FUNCTION_BLOCK FB_MonetTelescopeControl IMPLEMENTS I_Telescope
VAR_INPUT
(*
TCS interface section
see https://gitlab.aip.de/bmk10k/telescope_firmware/snippets/5
*)
	bPower				: BOOL;		// true: Power on, false: power off
	bGoHome				: BOOL;		// true: go to home position, unset track/goto if active
	bPark				: BOOL;		// boolean, true: go into park position, ready to stow telescope, unset track/goto
	bTrack				: BOOL;		// boolean, TRUE: MOVE telescope TO last ra/de AND start tracking. Set 'goto' TO FALSE, IF TRUE. FALSE: Stop tracking as soon as possible
	bGoto				: BOOL;		// boolean, TRUE: MOVE telescope TO tau/de AND stop there. Set track TO FALSE, IF TRUE. FALSE: no effect.)	
	bSlew				: BOOL;		// move the telescope to a given az-alt position
	bStop				: BOOL;		// boolean, TRUE: Stop motion OF telescope immediately, set goto AND track TO FALSE. FALSE: Allow motion OF telescope again via track/goto).	
	bReset				: BOOL;		// initiates reset on all axis
	bAutoTrack			: BOOL := TRUE;	// automatic tracking after goto
	fRightAscension		: LREAL := (4.0 + 35.0/60.0 + 54.09/3600.0) *15.0;	// apparent right ascension, degrees, double	
	fDeclination		: LREAL := 16.0 + 30.0/60.0 + 25.4/3600.0;	// apparent declination, degrees, double
	fElevation			: LREAL := 45.0;	// desired elevation of the telescope pointing
	fAzimuth			: LREAL := 320.0;	// desired azimut of the telescope pointing
	fElevationOffset	: LREAL := 0.0;		// absolute offset for elevation
	fAzimuthOffset 		: LREAL := 0.0;		// absolute offset for azimuth
	fTimeOffset			: LREAL := 0.0;		// absolute offset for time
	fDerotatorOffset	: LREAL := 0.0;		// offset for the de-rotator
	
	bEstopTriggered		: BOOL	:= FALSE;	// TODO: CHANGE
	bBrakeClearing		: BOOL	:= TRUE;
	bMainReady			: BOOL	:= TRUE;
	
	fbFocus				: I_Focus;
	fbCovers			: I_MirrorCovers;
	fbBrake				: I_Brake;	
	fbHydraulics   		: I_Hydraulics;
	fbElevation			: REFERENCE TO FB_ElevationControl;
	fbAzimuth			: REFERENCE TO FB_AzimuthControl;
	fbDerotator			: REFERENCE TO FB_DerotatorControl;

	telescopeConfig		: ST_TelescopeConfig;
END_VAR
VAR
	TelescopeAuxiliary	: FB_TelescopeAuxiliary;

	comm 				: I_Comm;
	
	TCS_command			: E_TCSCommand;	// actual command from the TCS
	jd					: LREAL;	// current Julian Date calculated from system time
	derotation_calc		: LREAL;	// image derotation
	lst					: LREAL;	// local siderial time calculated from Julian date
	fElevationInstr     : LREAL;
	fAzimuthInstr       : LREAL;
	fElevationPointing  : LREAL;
	fAzimuthPointing    : LREAL;
	fElevationCurrent   : LREAL;
	fAzimuthCurrent     : LREAL;
	fRAPointing         : LREAL;
	fDecPointing        : LREAL;
	elevation_calc		: LREAL;	// elevation calulated when ra and dec are set by TCS 
	azimuth_calc		: LREAL;	// azimuth calulated when ra and dec are set by TCS
	rightascension_calc	: LREAL;	// right ascension calulated when azimuth and elevation are set by TCS
	declination_calc	: LREAL;	// declination calulated when azimuth and elevation are set by TCS
	Hourangle_calc		: LREAL;	// hour angle
	fbTime				: FB_AstroClock;	// precise astronomical	time
	eq2hor				: FB_EQ2HOR;
	hor2eq				: FB_HOR2EQ;
	
	reset_trigger		: R_TRIG;
	
	powerfailure		: BOOL;		// triggers power-failure event
	poweronwarning		: TP;		// triggers power warning
	power_timeout		: TON;		// power on timeout
	command_timeout		: TON;		// command timeout
	tracking_delay		: TON;		// tracking delay
	isparked			: BOOL;		// telescope is parked
	TCSpowerEvent,
	TCSgohomeEvent,
	TCSparkEvent,
	TCSgotoEvent,
	TCStrackEvent,
	TCSstopEvent,
	AltitudeEvent,
	TCSreadyEvent,
	TCSCTOEvent			: FB_Eventlog;
	MQTTTimer 			: TON := (PT:=T#5S);
	
	DerotatorVelocity	: LREAL;	// rotational velocity of the derotator
	ElevationVelocity	: LREAL;	// rotational velocity of the elevation
	AzimuthVelocity		: LREAL;	// rotational velocity of the elevation
	derotatation_sign	: LREAL := 1.0;	// sign of derotation
	StatusWord, LastStatus:	UDINT;
END_VAR
VAR_OUTPUT
	bReady				: BOOL;		//		TRUE, IF telescope can be operated 
	bError				: BOOL;		// indicates an error on one of the components	
	errorid				: UDINT;	//error id of axis	
	bSliding				: BOOL;		//TRUE, IF telescope is in fast-MOVE phase (includes pole-swap)	
	bTracking			: BOOL;		//TRUE, IF telescope is on tracking position AND currently tracking.	
	bStopped				: BOOL;		//TRUE, IF telescope is AT rest.	
	elevation_current	: LREAL;	// true position of the elevation
	azimuth_current		: LREAL;	// true position of the azimuth
	derotator_current	: LREAL;	// true position of the de-rotator
	slewtime			: LREAL;	//	(time in sec. to reach the goto/track position) 
	bHomed				: BOOL;		// True: telescope is calibrated
	bBusy				: BOOL;		// telescope does not accept further commands
END_VAR
VAR PERSISTENT
	// elevation encoder zero offset
	EOFF:   LREAL;
	// azimuth axis offset/misalignment north-south
	AN_E:	LREAL;
	// azimuth axis offset/misalignment east-west
	AE_E:	LREAL;
	// gravitational flexure correction at the horizon
	TF:		LREAL;
	// azimuth encoder zero offset
	AOFF:   LREAL;
	// collimation error of the electromagnetic axis
	BNP:	LREAL;
	// azimuth axis offset/misalignment north-south
	AN_A:	LREAL;
	// azimuth axis offset/misalignment east-west,
	AE_A:	LREAL;
	// Non-perpendicularity between the mount azimuth and elevation axes
	NPAE:	LREAL;
END_VAR

TelescopeAuxiliary(comm := comm);

// get the system time
fbTime();
jd := DateTime2JD(fbTime.time_RTCEX2);
lst := CT2LST(telescopeConfig.longitude, jd);
// set reset state either by hardware (key pressed) or by software (set by e.g. tcs)
//IF GVL_Main.reset_switch THEN
	//reset := TRUE;
//END_IF

reset_trigger(CLK := bReset);

IF fbElevation.Error THEN
	errorid := fbElevation.nErrorID;
	fbElevation.bReset := bReset;
ELSIF fbAzimuth.bError THEN
	errorid := fbAzimuth.nErrorID;
	fbAzimuth.bReset := bReset;
ELSIF fbFocus <> 0 AND_THEN fbFocus.Error THEN
	errorid := fbFocus.ErrorID;
	IF reset_trigger.Q THEN
		fbFocus.Reset();
	END_IF
ELSIF fbDerotator.bError THEN
	errorid := fbDerotator.nErrorID;
	fbDerotator.bReset := bReset;
END_IF

bError := fbElevation.Error OR 
		 fbAzimuth.bError OR
		 (fbFocus <> 0 AND_THEN fbFocus.Error) OR
		 fbDerotator.bError;

slewtime := MAX(MAX(fbElevation.fSlewTime, fbAzimuth.fSlewTime), fbDerotator.fSlewTime);
			
IF bError THEN
	bGoHome := 	FALSE;
	bTrack := 	FALSE;
	bGoto := 	FALSE;
	bSlew := 	FALSE;
ELSE
	errorid := 0;
END_IF

IF fbElevation.bError THEN
	fbElevation.Enable := FALSE;
	fbAzimuth.Enable := FALSE;
	fbBrake.CloseBrake();
END_IF

eq2hor(
	ra := fRightAscension,
	dec := fDeclination,
	lon := telescopeConfig.longitude,
	lat := telescopeConfig.latitude,
	JD := jd + fTimeOffset,
	alt => elevation_calc,
	az => azimuth_calc,
	ha => hourangle_calc);

// apply pointing model
//elevation_calc := elevation_calc + PointingModelElevation(azimuth_calc, elevation_calc, EOFF + fElevationOffset, AN_E, AE_E, TF);
//azimuth_calc := azimuth_calc + PointingModelAzimuth(azimuth_calc, elevation_calc, AOFF + fAzimuthOffset, BNP, AN_A, AE_A, NPAE);
// calculate derotator position 
derotation_calc := F_DerotatorPosition2(azimuth_calc, elevation_calc, declination_calc, telescopeConfig.latitude, derotatation_sign)  + fDerotatorOffset;
// calculate velocities
DerotatorVelocity := F_Derotatorvelocity(elevation_calc, azimuth_calc, telescopeConfig.latitude);
ElevationVelocity := F_Elevationvelocity(azimuth_calc, telescopeConfig.latitude);
AzimuthVelocity := F_Azimuthvelocity(elevation_calc, azimuth_calc, telescopeConfig.latitude);

// calculate velocities
DerotatorVelocity := F_Derotatorvelocity(elevation_calc, azimuth_calc, telescopeConfig.latitude);
ElevationVelocity := F_Elevationvelocity(azimuth_calc, telescopeConfig.latitude);
AzimuthVelocity := F_Azimuthvelocity(elevation_calc, azimuth_calc, telescopeConfig.latitude);

IF (azimuth_calc > 310.0 AND AzimuthVelocity > 0.0) OR (azimuth_calc > 440.0) THEN
	azimuth_calc := azimuth_calc - 360.0;
ELSIF (azimuth_calc < 80.0 AND AzimuthVelocity < 0.0) OR (azimuth_calc < -50.0) THEN
	azimuth_calc := azimuth_calc + 360.0;
END_IF

IF (derotation_calc > 290.0 AND DerotatorVelocity > 0.0) OR (derotation_calc > 380.0) THEN
	derotation_calc := derotation_calc - 360.0;
ELSIF (derotation_calc < 20.0 AND DerotatorVelocity < 0.0) OR (derotation_calc < -70.0) THEN
	derotation_calc := derotation_calc + 360.0;
END_IF

// get current coordinates	
azimuth_current := fbAzimuth.fActualPosition;
elevation_current := fbElevation.fActualPosition;
derotator_current := fbDerotator.fActualPosition;

// apply pointing model
fElevationPointing := elevation_current - PointingModelElevation(azimuth_current, elevation_current, EOFF, AN_E, AE_E, TF);
fAzimuthPointing := azimuth_current - PointingModelAzimuth(azimuth_current, elevation_current, AOFF, BNP, AN_A, AE_A, NPAE);

// add offsets
fElevationCurrent := fElevationPointing - fElevationOffset;
fAzimuthCurrent := fAzimuthPointing - fAzimuthOffset;

// calculate equatorial coordinates
hor2eq(alt := fElevationCurrent, 
		az := fAzimuthCurrent,
		jd := jd,
		lat := telescopeConfig.latitude,
		lon := telescopeConfig.longitude,
		altitude := telescopeConfig.altitude,
		ra => rightascension_calc,
		dec => declination_calc);		
hor2eq(alt := fElevationPointing, 
		az := fAzimuthPointing,
		jd := jd,
		lat := telescopeConfig.latitude,
		lon := telescopeConfig.longitude,
		altitude := telescopeConfig.altitude,
		ra => fRAPointing,
		dec => fDecPointing);
	
poweronwarning(IN := bPower OR (NOT fbElevation.bEnable AND fbBrake.BrakeOpen), PT := T#250MS);

power_timeout(IN := TCS_command = E_TCSCommand.no_command AND NOT isparked, PT := T#12H);
command_timeout();
IF power_timeout.Q AND NOT isparked THEN
	bPark := TRUE;
END_IF
		
// set TCS_command according to state variables ordered by precedence
IF bPower THEN
	TCS_command := E_TCSCommand.poweron;
ELSIF bStop THEN
	TCS_command := E_TCSCommand.stop;
	bGoto := FALSE;
	bTrack := FALSE;
	bSlew := FALSE;
	bGoHome := FALSE;
	bPark := FALSE;
ELSIF bPark THEN
	bGoto := FALSE;
	bTrack := FALSE;
	bSlew := FALSE;
	IF bReady AND bStopped THEN
		TCS_command := E_TCSCommand.park;
	END_IF
ELSIF bGoHome THEN
	bGoto := FALSE;
	bTrack := FALSE;
	bSlew := FALSE;
	IF bReady AND NOT bBusy AND bStopped THEN
		TCS_command := E_TCSCommand.gohome;
	END_IF
ELSIF bGoto THEN
	bTrack := FALSE;
	bSlew := FALSE;
	IF bReady AND NOT bBusy THEN
		TCS_command := E_TCSCommand.goto;
	END_IF
ELSIF bSlew THEN
	bGoto := FALSE;
	bTrack := FALSE;
	IF bReady AND NOT bBusy THEN
		TCS_command := E_TCSCommand.slew;
	END_IF
ELSIF bTrack THEN
	bGoto := FALSE;
	bSlew := FALSE;
	IF bReady AND NOT bBusy THEN
		TCS_command := E_TCSCommand.track;
	END_IF
ELSE
	TCS_command := E_TCSCommand.no_command;
	fbElevation.bMoveAxis := FALSE;
	fbAzimuth.bMoveAxis := FALSE;
	fbDerotator.bMoveAxis := FALSE;
	fbElevation.bTracking := FALSE;
	fbAzimuth.bTracking := FALSE;
	fbDerotator.bTracking := FALSE;
END_IF

IF TCS_command = E_TCSCommand.poweron THEN
	_PowerOn();
	command_timeout(IN := TCS_command = E_TCSCommand.poweron, PT := T#12H);
	TCSCTOEvent.OnMessage := 'POWER';
ELSIF TCS_command = E_TCSCommand.stop THEN
	_StopTelescope();
	command_timeout(IN := TCS_command = E_TCSCommand.stop, PT := T#2S);
	TCSCTOEvent.OnMessage := 'STOP';
ELSIF TCS_command = E_TCSCommand.park THEN
	_ParkTelescope();
	command_timeout(IN := TCS_command = E_TCSCommand.park, PT := T#2M);
	TCSCTOEvent.OnMessage := 'PARK';
ELSIF TCS_command = E_TCSCommand.gohome THEN
	_HomeTelescope();
	command_timeout(IN := TCS_command = E_TCSCommand.gohome, PT := T#2M);
	TCSCTOEvent.OnMessage := 'GOHOME';
ELSIF TCS_command = E_TCSCommand.goto THEN
	_GotoTelescope();
	command_timeout(IN := TCS_command = E_TCSCommand.goto, PT := T#2M);
	TCSCTOEvent.OnMessage := 'GOTO';
ELSIF TCS_command = E_TCSCommand.slew THEN
	_SlewTelescope();
	command_timeout(IN := TCS_command = E_TCSCommand.slew, PT := T#2M);
	TCSCTOEvent.OnMessage := 'SLEW';
ELSIF TCS_command = E_TCSCommand.track THEN
	_TrackTelescope();
	command_timeout(IN := TCS_command = E_TCSCommand.track, PT := T#12H);
	TCSCTOEvent.OnMessage := 'TRACK';
ELSE
	// disable command timeout
	command_timeout(IN := FALSE);
	TCSCTOEvent.OnMessage := 'NOCOMMAND';
END_IF
 
bSliding := NOT bTracking AND (fbElevation.fbAxis.InMotion OR fbElevation.fbAxis.InRamp OR
			fbAzimuth.fbAxis.InMotion OR fbAzimuth.fbAxis.InRamp OR
			fbDerotator.fbAxis.InMotion OR fbDerotator.fbAxis.InRamp);

// signal must be stable for 5500MS
tracking_delay(in := fbElevation.fbAxis.isTracking AND 
			fbAzimuth.fbAxis.isTracking AND
			fbDerotator.fbAxis.isTracking,PT :=T#5500MS, Q => bTracking);
			
bStopped :=  (NOT fbElevation.bEnable OR fbElevation.fbAxis.StandStill) AND 
			(NOT fbAzimuth.bEnable OR fbAzimuth.fbAxis.StandStill) AND
			(NOT fbDerotator.bEnable OR fbDerotator.fbAxis.StandStill);
			
bHomed := fbElevation.bCalibrated AND
			fbAzimuth.bCalibrated AND
			fbDerotator.bCalibrated;
IF fbFocus <> 0 THEN
	bHomed := bHomed AND fbFocus.Calibrated;
END_IF
			
bReady := bHomed AND 
	fbCovers.Opened AND 
	fbElevation.bEnable AND
	fbAzimuth.bEnable AND
	fbDerotator.bEnable AND fbBrake.BrakeOpen AND 
    NOT bError;

bBusy := fbElevation.fbAxis.Busy OR
		fbAzimuth.fbAxis.Busy OR
		fbDerotator.fbAxis.Busy;
IF fbFocus <> 0 THEN
	bBusy := bBusy AND fbFocus.Busy;
END_IF		

// unset the STOP command if telescope is already stopped
IF bStopped THEN
	bStop := FALSE;
END_IF
	
IF NOT bError THEN
	bReset := FALSE;
END_IF

IF bEstopTriggered THEN
	fbElevation.Enable := FALSE;
	fbAzimuth.Enable := FALSE;
	fbDerotator.Enable := FALSE;
END_IF
IF bSliding OR bTrack OR bTracking THEN
	MQTTTimer.PT := T#1000MS;
ELSE
	MQTTTimer.PT := T#5000MS;
END_IF
MQTTTimer(IN:=TRUE);
IF MQTTTimer.Q THEN // publish new payload every second
	MQTTTimer(IN:=FALSE);

	comm.Publish('telescope', 'dome', 'JulianDate', LREAL_TO_STRING(jd));
	comm.Publish('telescope', 'dome', 'LocalSiderialTime', LREAL_TO_STRING(lst));
	comm.Publish('telescope', 'dome', 'Azimuth', LREAL_TO_STRING(azimuth_current));
	comm.Publish('telescope', 'dome', 'Elevation', LREAL_TO_STRING(elevation_current));
	comm.Publish('telescope', 'dome', 'Derotator', LREAL_TO_STRING(derotator_current));
	comm.Publish('telescope', 'dome', 'HourAngle', LREAL_TO_STRING(hourangle_calc));
	//comm.Publish('telescope', 'dome', 'RightAscension', LREAL_TO_STRING(rightascension_calc));
	//comm.Publish('telescope', 'dome', 'Declination', LREAL_TO_STRING(declination_calc));
	comm.Publish('telescope', 'dome', 'RightAscension', LREAL_TO_STRING(fRightAscension));
	comm.Publish('telescope', 'dome', 'Declination', LREAL_TO_STRING(fDeclination));
	comm.Publish('telescope', 'dome', 'azimuth_offset', LREAL_TO_STRING(fAzimuthOffset));
	comm.Publish('telescope', 'dome', 'elevation_offset', LREAL_TO_STRING(fElevationOffset));
	comm.Publish('telescope', 'dome', 'derotator_torque', LREAL_TO_STRING(fbDerotator.fTorque));
	comm.Publish('telescope', 'dome', 'elevation_torque', LREAL_TO_STRING(fbElevation.fTorque));
	comm.Publish('telescope', 'dome', 'azimuth_torque', LREAL_TO_STRING(fbAzimuth.fTorque));
	
	comm.Publish('telescope', 'dome', 'errorid',		UDINT_TO_STRING(errorid));
	comm.Publish('telescope', 'dome', 'error',		BOOL_TO_STRING(bError));
	comm.Publish('telescope', 'dome', 'ready',		BOOL_TO_STRING(bReady));
	comm.Publish('telescope', 'dome', 'busy',		BOOL_TO_STRING(bBusy));
	comm.Publish('telescope', 'dome', 'sliding',		BOOL_TO_STRING(bSliding));
	comm.Publish('telescope', 'dome', 'tracking', 	BOOL_TO_STRING(bTracking));
	comm.Publish('telescope', 'dome', 'stopped',		BOOL_TO_STRING(bStopped));
	comm.Publish('telescope', 'dome', 'homed',		BOOL_TO_STRING(bHomed));
	comm.Publish('telescope', 'dome', 'parked',		BOOL_TO_STRING(isparked));
	
	comm.Publish('telescope', 'dome', 'POSITION.INSTRUMENTAL.AZ.REALPOS', LREAL_TO_STRING(azimuth_current));
	comm.Publish('telescope', 'dome', 'POSITION.INSTRUMENTAL.AZ.OFFSET', LREAL_TO_STRING(fAzimuthOffset));
	comm.Publish('telescope', 'dome', 'POSITION.INSTRUMENTAL.ALT.REALPOS', LREAL_TO_STRING(elevation_current));
	comm.Publish('telescope', 'dome', 'POSITION.INSTRUMENTAL.ALT.OFFSET', LREAL_TO_STRING(fElevationOffset));	
	comm.Publish('telescope', 'dome', 'POSITION.CURRENT.AZ', LREAL_TO_STRING(fAzimuthPointing));
	comm.Publish('telescope', 'dome', 'POSITION.CURRENT.ALT', LREAL_TO_STRING(fElevationPointing));
	comm.Publish('telescope', 'dome', 'POSITION.CURRENT.RA', LREAL_TO_STRING(fRAPointing));
	comm.Publish('telescope', 'dome', 'POSITION.CURRENT.DEC', LREAL_TO_STRING(fDecPointing));
	comm.Publish('telescope', 'dome', 'POSITION.REAL.AZ', LREAL_TO_STRING(fAzimuthCurrent));
	comm.Publish('telescope', 'dome', 'POSITION.REAL.ALT', LREAL_TO_STRING(fElevationCurrent));

END_IF

StatusWord.0 := bError;
StatusWord.1 := bReady;
StatusWord.2 := bSliding;
StatusWord.3 := bTracking;
StatusWord.4 := bStopped;
StatusWord.5 := bHomed;
StatusWord.6 := bPower;
StatusWord.7 := bPark;
StatusWord.8 := bGoHome;
StatusWord.9 := bTrack;
StatusWord.10 := bGoto;
StatusWord.11 := bSlew;
StatusWord.12 := bStop;
StatusWord.13 := bBusy;

IF StatusWord<>LastStatus THEN // publish new payload every second
	LastStatus := StatusWord;
	comm.Publish('telescope', 'dome', 'error',		BOOL_TO_STRING(bError));
	comm.Publish('telescope', 'dome', 'ready',		BOOL_TO_STRING(bReady));
	comm.Publish('telescope', 'dome', 'sliding',		BOOL_TO_STRING(bSliding));
	comm.Publish('telescope', 'dome', 'tracking', 	BOOL_TO_STRING(bTracking));
	comm.Publish('telescope', 'dome', 'stopped',		BOOL_TO_STRING(bStopped));
	comm.Publish('telescope', 'dome', 'homed',		BOOL_TO_STRING(bHomed));
	comm.Publish('telescope', 'dome', 'power',		BOOL_TO_STRING(bPower));
	comm.Publish('telescope', 'dome', 'park',		BOOL_TO_STRING(bPark));
	comm.Publish('telescope', 'dome', 'gohome',		BOOL_TO_STRING(bGoHome));
	comm.Publish('telescope', 'dome', 'track',		BOOL_TO_STRING(bTrack));
	comm.Publish('telescope', 'dome', 'goto',		BOOL_TO_STRING(bGoto));
	comm.Publish('telescope', 'dome', 'slew',		BOOL_TO_STRING(bSlew));
	comm.Publish('telescope', 'dome', 'stop',		BOOL_TO_STRING(bStop));
	comm.Publish('telescope', 'dome', 'busy',		BOOL_TO_STRING(bBusy));
END_IF


(* Event function blocks start here. *)
TCSpowerEvent(	Trigger := powerfailure, 
				Level := ADSLOG_MSGTYPE_ERROR,
				FormatString := 'power %s',
				//OnMessage := 'Failure',
				OffMessage := 'OK', 
				Comm := comm);

TCSgohomeEvent(	Trigger := bGoHome, 
				Level := ADSLOG_MSGTYPE_HINT,
				FormatString := 'GOHOME %s',
				OnMessage := 'commencing',
				OffMEssage := 'completed', 
				Comm := comm);
TCSparkEvent(	Trigger := bPark, 
				Level := ADSLOG_MSGTYPE_HINT,
				FormatString := 'PARK %s',
				OnMessage := 'commencing',
				OffMEssage := 'completed', 
				Comm := comm);
TCSgotoEvent(	Trigger := bGoto, 
				Level := ADSLOG_MSGTYPE_HINT,
				FormatString := 'GOTO %s',
				OnMessage := 'commencing',
				OffMEssage := 'completed', 
				Comm := comm);
TCStrackEvent(	Trigger := bTrack, 
				Level := ADSLOG_MSGTYPE_HINT,
				FormatString := 'TRACK %s',
				OnMessage := 'commencing',
				OffMEssage := 'completed', 
				Comm := comm);
TCSstopEvent(	Trigger := bStop, 
				Level := ADSLOG_MSGTYPE_WARN,
				FormatString := 'STOP %s',
				OnMessage := 'commencing',
				OffMEssage := 'completed',
				OffLevel := ADSLOG_MSGTYPE_HINT, 
				Comm := comm);
AltitudeEvent(	Trigger := bPower AND elevation_calc<0.0, 
				Level := ADSLOG_MSGTYPE_WARN,
				FormatString := '%s',
				OnMessage := 'Target below horizon',
				OffMEssage := '', 
				Comm := comm);
TCSreadyEvent(	Trigger := bPower AND bReady, 
				Level := ADSLOG_MSGTYPE_HINT,
				FormatString := '%s',
				OnMessage := 'STELLA1 startup finished', 
				Comm := comm);
TCSCTOEvent(	Trigger := command_timeout.Q,
				Level := ADSLOG_MSGTYPE_WARN,
				FormatString := 'A timeout occured during %s command!',
				OnMessage := 'NOCOMMAND', 
				Comm := comm);

METHOD PRIVATE _GotoTelescope : USINT
VAR_INPUT
END_VAR
VAR
	GoToEvent		: FB_Eventlog;
	commandTimeout	: TON;
END_VAR
VAR_STAT
	Stage			: USINT := 0;
	LastStage		: USINT := 101;
END_VAR
_GotoTelescope := Stage;
commandTimeout(IN := Stage < 100, PT := T#600S);
IF commandTimeout.Q THEN
	bError := TRUE;
	errorid := 16#10;
	bGoto := FALSE;
	Stage := 0;
	RETURN;
END_IF

IF elevation_calc<2.0 THEN
	bError := TRUE;
	errorid := 16#15;
	bGoto := FALSE;
	Stage := 0;
	RETURN;
END_IF

IF bReset OR bError THEN
	Stage := 0;
	RETURN;
END_IF

CASE Stage OF
	0:	
		IF bReady AND NOT bBusy THEN
			Stage := 25;
		END_IF
	25:	
		fbElevation.Position := elevation_calc;
		fbAzimuth.Position := azimuth_calc;
		fbDerotator.Position := derotation_calc;
		fbDerotator.Velocity := 10.0;
		fbElevation.Velocity := 10.0;
		fbAzimuth.Velocity := 10.0;
		
		fbElevation.MoveAxis := TRUE;
		fbAzimuth.MoveAxis := TRUE;
		fbDerotator.MoveAxis := TRUE;
		IF fbElevation.Busy AND
			fbAzimuth.Busy AND
			fbDerotator.Busy THEN
				Stage := 50;
		END_IF
	50:
		IF NOT fbElevation.Busy AND fbElevation.MoveDone THEN
			fbElevation.MoveAxis := FALSE;
		END_IF
		IF NOT fbAzimuth.Busy AND fbAzimuth.MoveDone THEN
			fbAzimuth.MoveAxis := FALSE;
		END_IF
		IF NOT fbDerotator.Busy AND fbDerotator.MoveDone THEN
			fbDerotator.MoveAxis := FALSE;
		END_IF
		IF NOT fbElevation.MoveAxis AND 
           NOT fbAzimuth.MoveAxis AND 
		   NOT fbDerotator.MoveAxis THEN
		   Stage := 75;
		END_IF
	75:
		IF NOT bSliding AND bStopped THEN // all axis standstill
			Stage := 100;
		END_IF
	100:
		fbElevation.MoveAxis := FALSE;
		fbAzimuth.MoveAxis := FALSE;
		fbDerotator.MoveAxis := FALSE;
		fAzimuth := azimuth_calc;
		fElevation := elevation_calc;
		bGoto := FALSE;
		// enable automatic tracking
		bTrack := bAutoTrack;
		Stage := 0;
END_CASE
GoToEvent(Trigger := Stage > LastStage, FormatString := 'GoTo progress: %s', OnMessage := USINT_TO_STRING(Stage), comm := comm);
LastStage := Stage;
END_METHOD

METHOD PRIVATE _HomeTelescope : BOOL
VAR_INPUT
END_VAR
VAR
	HomeEvent		: FB_Eventlog;
	commandTimeout	: TON;
END_VAR
commandTimeout(IN := NOT _HomeTelescope, PT := T#600S);
IF commandTimeout.Q THEN
	bError := TRUE;
	errorid := 16#30;
	_HomeTelescope :=TRUE;
END_IF

IF bReady AND bStopped AND NOT bBusy AND NOT bTracking THEN
	fbElevation.Velocity := 10.0;
	fbElevation.Position := telescopeConfig.elevationHome;
	fbElevation.MoveAxis := TRUE;
	fbAzimuth.Velocity := 10.0;
	fbAzimuth.Position := telescopeConfig.azimuthHome;
	fbAzimuth.MoveAxis := TRUE;
	fbDerotator.Velocity := 10.0;
	fbDerotator.Position := telescopeConfig.derotatorHome;
	fbDerotator.MoveAxis := TRUE;	
END_IF

IF fbElevation.MoveDone AND 
	fbAzimuth.MoveDone AND 
	fbDerotator.MoveDone THEN
	bGoHome := FALSE;
	fElevation := elevation_current;
	fAzimuth := azimuth_current;
	_HomeTelescope := TRUE;
ELSE
	_HomeTelescope := FALSE;
END_IF

HomeEvent(Trigger := _HomeTelescope, 
			Level := ADSLOG_MSGTYPE_HINT,
			FormatString := '%s',
			OnMessage := 'Telescope is homed.', comm := comm);
END_METHOD

METHOD PRIVATE _ParkTelescope : USINT
VAR_INPUT
END_VAR
VAR
	ParkEvent	: FB_Eventlog;
END_VAR
VAR_STAT
	Stage		: USINT := 0;
	LastStage	: USINT := 101;
END_VAR
_ParkTelescope := Stage;
IF bReset OR bError THEN
	Stage := 0;
END_IF
IF isparked THEN
	Stage := 100;
END_IF
CASE Stage OF
	0: 
		bGoHome := 	FALSE;
		bTrack := 	FALSE;
		bGoto := 	FALSE;
		bSlew := 	FALSE;
		IF fbFocus <> 0 THEN
			fbFocus.Position := telescopeConfig.focusPark;
		END_IF
		IF bError THEN // emergency park
			fbBrake.CloseBrake();
			fbElevation.Enable := FALSE;
			fbAzimuth.Enable := FALSE;
			fbDerotator.Enable := FALSE;	
			fbCovers.Close();	
			Stage := 80;
		END_IF
		Stage := 20;
	20:
		fbElevation.Position := telescopeConfig.elevationPark;
		fbElevation.Velocity := 10.0;
		fbElevation.MoveAxis := TRUE;
		fbAzimuth.Position := telescopeConfig.azimuthPark;
		fbAzimuth.Velocity := 10;
		fbAzimuth.MoveAxis := TRUE;
		fbDerotator.Position := telescopeConfig.derotatorPark;
		fbDerotator.Velocity := 10.0;
		fbDerotator.MoveAxis := TRUE;
		IF fbElevation.Busy AND
			fbAzimuth.Busy AND
			fbDerotator.Busy THEN
				Stage := 40;
		END_IF
	40:
		IF fbElevation.MoveDone THEN
			fbElevation.MoveAxis := FALSE;
		END_IF
		IF fbAzimuth.MoveDone THEN
			fbAzimuth.MoveAxis := FALSE;
		END_IF
		IF fbDerotator.MoveDone THEN
			fbDerotator.MoveAxis := FALSE;
		END_IF
		IF NOT bSliding THEN // all axis standstill
			Stage := 60;
		END_IF
	60:
		IF NOT fbElevation.Enable AND NOT fbAzimuth.Enable AND NOT fbDerotator.Enable THEN
			stage := 80;
		END_IF

		IF bStopped THEN
			fbElevation.Enable := FALSE;
			fbAzimuth.Enable := FALSE;
			fbDerotator.Enable := FALSE;
		END_IF
		
		fbElevation.bMoveAxis := FALSE;
		fbAzimuth.bMoveAxis := FALSE;
		fbDerotator.bMoveAxis := FALSE;
	80:
		IF fbElevation.Enable OR fbAzimuth.Enable OR fbDerotator.Enable THEN
			stage := 60;
		END_IF
		IF NOT fbBrake.BrakeOpen THEN
			fbCovers.Close();
			fbHydraulics.Enable := FALSE;
		END_IF
		IF fbCovers.Closed THEN
			Stage := 100;
		END_IF
	100:
			isparked := TRUE;
			bPark := FALSE;
			_ParkTelescope := 100;
			Stage := 0;	
END_CASE
ParkEvent(Trigger := Stage > LastStage, FormatString := 'Parking progress: %s', OnMessage := USINT_TO_STRING(Stage), comm := comm);
LastStage := Stage;
END_METHOD

METHOD PRIVATE _PowerOn : BOOL
VAR_INPUT
END_VAR
IF NOT bBrakeClearing THEN
	powerfailure := TRUE;
	TCSpowerEvent.OnMessage := 'failure: brake clearing not set';
	bPower := FALSE;
ELSIF bError THEN
	powerfailure := TRUE;
	TCSpowerEvent.OnMessage := 'Generic error during power on occured.';
	bPower := FALSE;
ELSE
	powerfailure := FALSE;		
END_IF
// COVER MUST BE OPENED FOR A SUCCESSFUL WAKE & SHAKE COMMAND!
fbCovers.Open();

// enable elevation, enable azimuth
IF bMainReady AND fbCovers.Opened THEN
	fbElevation.Enable := TRUE;
	fbAzimuth.Enable := TRUE;
	fbDerotator.Enable := TRUE;
END_IF

IF fbElevation.Ready AND NOT fbElevation.Calibrated THEN
	fbElevation.HomeAxis := TRUE;
END_IF

IF fbAzimuth.Ready AND NOT fbAzimuth.Calibrated THEN
	fbAzimuth.HomeAxis := TRUE;
END_IF

// enable derotator
IF fbElevation.Ready THEN
	fbDerotator.HomeAxis := fbDerotator.Ready AND NOT fbDerotator.Calibrated;
END_IF

// start calibration of focus after elevation has been calibrated
// this avoids imbalance by the M2 mirror on the elvation during its calibration
IF fbElevation.Calibrated AND (fbFocus <> 0 AND_THEN NOT fbFocus.Calibrated) THEN
	fbFocus.Enable := TRUE;
	fbFocus.HomeAxis := TRUE;
END_IF

IF fbCovers.Opened AND 
	fbElevation.Calibrated AND
	fbAzimuth.Calibrated AND
	fbDerotator.Calibrated THEN
	//FocusControl.Calibrated THEN
	bPower := FALSE;
	_PowerOn := TRUE;
	isparked := FALSE;
	// slew the telescope to the home position
	bGoHome := TRUE;
ELSE
	_PowerOn := FALSE;
END_IF
END_METHOD

METHOD PRIVATE _SlewTelescope : USINT
VAR_INPUT
END_VAR
VAR
	SlewEvent:	FB_Eventlog;
	command_timeout: TON;
END_VAR
VAR_STAT
	Stage:		USINT := 0;
	LastStage:	USINT := 101;
END_VAR
_SlewTelescope := Stage;
command_timeout(IN := Stage < 100, PT := T#600S);
IF command_timeout.Q THEN
	bError := TRUE;
	errorid := 16#40;
	bSlew := FALSE;
	Stage := 0;
END_IF
IF bReset OR bError THEN
	Stage := 0;
END_IF
CASE Stage OF
	0:	
		IF bReady AND bStopped AND NOT bBusy AND NOT bTracking THEN
			Stage := 25;
		END_IF
	25:
		fbElevation.Position := fElevation + PointingModelElevation(fAzimuth, fElevation, EOFF + fElevationOffset, AN_E, AE_E, TF);
		fbElevation.Velocity := 10.0;
		fbElevation.MoveAxis := TRUE;
		fbAzimuth.Position := fAzimuth + PointingModelAzimuth(fAzimuth, fElevation, AOFF + fAzimuthOffset, BNP, AN_A, AE_A, NPAE);
		fbAzimuth.Velocity := 10.0;
		fbAzimuth.MoveAxis := TRUE;
		fbDerotator.Position := fElevation + fDerotatorOffset;
		fbDerotator.Velocity := 10.0;
		fbDerotator.MoveAxis := TRUE;
		IF fbElevation.Busy AND
			fbAzimuth.Busy AND
			fbDerotator.Busy THEN
				Stage := 50;
		END_IF
	50:
		IF fbElevation.MoveDone THEN
			fbElevation.bMoveAxis := FALSE;
		END_IF
		
		IF fbAzimuth.MoveDone THEN
			fbAzimuth.MoveAxis := FALSE;
		END_IF

		IF fbDerotator.MoveDone THEN
			fbDerotator.MoveAxis := FALSE;
		END_IF
		IF NOT bSliding AND bStopped THEN // all axis standstill
			Stage := 100;
		END_IF
	100:
		fbElevation.MoveAxis := FALSE;
		fbAzimuth.MoveAxis := FALSE;
		fbDerotator.MoveAxis := FALSE;
		fRightAscension := rightascension_calc;
		fDeclination := declination_calc;
		bSlew := FALSE;
		Stage := 0;
END_CASE
SlewEvent(Trigger := Stage > LastStage, FormatString := 'Slew progress: %s', OnMessage := USINT_TO_STRING(Stage), comm := comm);
LastStage := Stage;
END_METHOD

METHOD PRIVATE _StopTelescope : BOOL
VAR_INPUT
END_VAR
fbElevation.StopAxis := TRUE;
fbAzimuth.StopAxis := TRUE;
fbDerotator.StopAxis := TRUE;
IF bStopped THEN
	fbElevation.StopAxis := FALSE;
	fbAzimuth.StopAxis := FALSE;
	fbDerotator.StopAxis := FALSE;
	_StopTelescope := FALSE;
END_IF
END_METHOD

METHOD PRIVATE _TrackTelescope : BOOL
VAR_INPUT
END_VAR
// Elevation
DerotatorVelocity := F_Derotatorvelocity(elevation_calc, azimuth_calc, telescopeConfig.latitude);
ElevationVelocity := F_Elevationvelocity(azimuth_calc, telescopeConfig.latitude);
AzimuthVelocity := F_Azimuthvelocity(elevation_calc, azimuth_calc, telescopeConfig.latitude);
IF elevation_current < 5.0 OR elevation_current > 89.5 THEN 
	bTrack := FALSE;
END_IF
IF azimuth_current > 440.0 THEN
	bTrack := FALSE;
END_IF
IF (derotator_current < -69.0 AND DerotatorVelocity<0.0) OR (derotator_current > 379.0 AND DerotatorVelocity>0.0) THEN
	bTrack := FALSE;
END_IF

fbElevation.Position := elevation_calc;
IF NOT fbElevation.Tracking THEN
	fbElevation.Velocity := 10.0;
	fbElevation.MoveAxis := TRUE;
	IF NOT fbElevation.Busy AND fbElevation.MoveDone THEN
		fbElevation.MoveAxis := FALSE;
		IF fbElevation.isTracking THEN
			fbElevation.Velocity := ElevationVelocity;
		ELSE
			fbElevation.Velocity := 3.0*ElevationVelocity;
		END_IF
		fbElevation.Velocity := ElevationVelocity;
		fbElevation.Tracking := TRUE;
	END_IF
ELSE
	fbElevation.Velocity := ElevationVelocity;
END_IF

// Azimuth
fbAzimuth.Position := azimuth_calc;
IF NOT fbAzimuth.Tracking THEN
	fbAzimuth.Velocity := 10.0;
	fbAzimuth.MoveAxis := TRUE;
	IF NOT fbAzimuth.Busy AND fbAzimuth.MoveDone THEN
		fbAzimuth.MoveAxis := FALSE;
		IF fbAzimuth.isTracking THEN
			fbAzimuth.Velocity := AzimuthVelocity;
		ELSE
			fbAzimuth.Velocity := 3.0*AzimuthVelocity;
		END_IF
		fbAzimuth.Velocity := AzimuthVelocity;
		fbAzimuth.Tracking := TRUE;
	END_IF
ELSE
	fbAzimuth.Velocity := AzimuthVelocity;
END_IF

// Derotator
fbDerotator.Position := derotation_calc;
IF NOT fbDerotator.Tracking THEN
	fbDerotator.Velocity := 10.0;
	fbDerotator.MoveAxis := TRUE;
	IF NOT fbDerotator.Busy AND fbDerotator.MoveDone THEN
		fbDerotator.MoveAxis := FALSE;
		IF fbDerotator.isTracking THEN
			fbDerotator.Velocity := DerotatorVelocity;
		ELSE
			fbDerotator.Velocity := 3.0*DerotatorVelocity;
		END_IF
		fbDerotator.Velocity := DerotatorVelocity;
		fbDerotator.Tracking := TRUE;
	END_IF
ELSE
	fbDerotator.Velocity := DerotatorVelocity;
END_IF
END_METHOD

{warning 'add property implementation'}
PROPERTY Altitude : LREAL
GET
Altitude := THIS^.fElevationCurrent;
END_GET
END_PROPERTY

{warning 'add property implementation'}
PROPERTY Azimuth : LREAL
GET
Azimuth := THIS^.fAzimuthCurrent;
END_GET
END_PROPERTY

{warning 'add property implementation'}
PROPERTY Declination : LREAL
GET
Declination := THIS^.fDeclination;
END_GET
END_PROPERTY

//FB_Init is always available implicitly and it is used primarily for initialization.
//The return value is not evaluated. For a specific influence, you can also declare the
//methods explicitly and provide additional code there with the standard initialization
//code. You can evaluate the return value.
METHOD FB_Init: BOOL
VAR_INPUT
    bInitRetains	: BOOL; // TRUE: the retain variables are initialized (reset warm / reset cold)
    bInCopyCode		: BOOL;  // TRUE: the instance will be copied to the copy code afterward (online change)
	comm			: I_Comm;
END_VAR
THIS^.comm 				:= comm;
END_METHOD

METHOD Home : BOOL
bGoHome := TRUE;
END_METHOD

METHOD Init : BOOL
bPower := TRUE;
END_METHOD

METHOD MoveAltAz : BOOL
VAR_INPUT
	AltAz	: BROTLib.ST_AltAzCoordinate;
END_VAR
fElevation 	:= AltAz.Altitude;
fAzimuth 	:= AltAz.Azimuth;
bSlew		:= TRUE;
END_METHOD

METHOD MoveRaDec : BOOL
VAR_INPUT
	RaDec	: BROTLib.ST_RaDecCoordinate;
END_VAR
fRightAscension	:= RaDec.RightAscension;
fDeclination	:= RaDec.Declination;
bGoto			:= TRUE;
END_METHOD

METHOD Park : BOOL
bPark := TRUE;
END_METHOD

METHOD Reset : BOOL
bReset := TRUE;
END_METHOD

{warning 'add property implementation'}
PROPERTY RightAscension : LREAL
GET
RightAscension := THIS^.fRightAscension;
END_GET
END_PROPERTY

METHOD SetAltitudeOffset : BOOL
VAR_INPUT
	Offset	: LREAL;
END_VAR
fElevationOffset := Offset;
END_METHOD

METHOD SetAzimuthOffset : BOOL
VAR_INPUT
	Offset	: LREAL;
END_VAR
fAzimuthOffset := Offset;
END_METHOD

METHOD SetDerotatorOffset : BOOL
VAR_INPUT
	Offset	: LREAL;
END_VAR
fDerotatorOffset := Offset;
END_METHOD

{warning 'add method implementation '}
METHOD Slew : BOOL
VAR_INPUT
	fAzimuth	: LREAL;
	fAltitude	: LREAL;
END_VAR
THIS^.fElevation 	:= fAltitude;
THIS^.fAzimuth 	:= fAzimuth;
THIS^.bSlew		:= TRUE;
END_METHOD

METHOD Stop : BOOL
bStop := TRUE;
END_METHOD

{warning 'add method implementation '}
METHOD Track : BOOL
VAR_INPUT
	fRightAscension	: LREAL;
	fDeclination	: LREAL;
END_VAR
THIS^.fRightAscension	:= fRightAscension;
THIS^.fDeclination		:= fDeclination;
THIS^.bTrack			:= TRUE;
END_METHOD

METHOD TrackRaDec : BOOL
VAR_INPUT
	RaDec	: BROTLib.ST_RaDecCoordinate;
END_VAR
fRightAscension	:= RaDec.RightAscension;
fDeclination		:= RaDec.Declination;
bTrack			:= TRUE;
END_METHOD

END_FUNCTION_BLOCK

(* stored: Version 1.1.0.1, ProductVersion 3.1.4024.15
   POU FB_MonetTelescopeControl: Id {10c2c294-efcf-424f-afd3-75ac57a5e8bc}, SpecialFunc None
   Method _GotoTelescope: Id {43ebaf76-c0fc-41db-8c98-2f7671dc6b31}
   Method _HomeTelescope: Id {b2d9dfb4-bf7c-4f17-8ac5-7f074d6808c9}
   Method _ParkTelescope: Id {94a12771-4c75-4743-9ad3-850f66878f1f}
   Method _PowerOn: Id {1dafa267-4251-4a45-a8e2-ae0ece289894}
   Method _SlewTelescope: Id {4aaca2e7-2dba-4c2d-80b3-cd4dcc5ad38b}
   Method _StopTelescope: Id {cc9583d1-2578-4480-8aee-f6d55f373bf1}
   Method _TrackTelescope: Id {0dd53d55-2f74-4268-9438-8bb832d1c59b}
   Property Altitude: Id {08036c9a-29a6-4dff-81c5-9c4ffdbe1388}
   Get Get: Id {69f2fe63-a318-4eda-9ea8-726f0beaaa1a}
   Property Azimuth: Id {c361ba59-5813-4434-a60f-689a4e8b98db}
   Get Get: Id {1a2b67ba-bdac-4452-819a-ecc849847788}
   Property Declination: Id {dbc97a9f-600a-4687-aad4-75127caee214}
   Get Get: Id {e9074fb4-1eac-44d4-af03-6b3c48c41fa7}
   Method FB_Init: Id {034c34d9-521a-4d54-9624-e4d1bdeb670c}
   Method Home: Id {1ffeeb7f-e086-4ec6-b333-bf9ff24723c8}
   Method Init: Id {a631cabc-b5f9-4584-b7df-b1ee9d39f6ec}
   Method MoveAltAz: Id {c6c43861-5da1-4194-b463-81c0490ebb78}
   Method MoveRaDec: Id {f860f1af-1ff9-4d1a-a407-9f1e7e899f51}
   Method Park: Id {d8a2b837-9b51-4592-a9b7-5ddb1b1403bd}
   Method Reset: Id {f3acfef0-ab57-4326-aaf5-f5730beeec6a}
   Property RightAscension: Id {73651e6e-c817-4911-a062-89ad8486672a}
   Get Get: Id {e6187f66-c4f4-4ea1-b2f6-82d1dac4a0b4}
   Method SetAltitudeOffset: Id {10a7c758-0667-41d2-90bb-38e90ad006bf}
   Method SetAzimuthOffset: Id {f9c99137-b576-45ed-a746-cd632ae8760e}
   Method SetDerotatorOffset: Id {4346176d-5ecc-4074-804b-bfb36ac0210a}
   Method Slew: Id {97a8c7d7-3c79-4306-b601-6d1789eff988}
   Method Stop: Id {e66d844d-991d-4af1-8b55-fe6740342385}
   Method Track: Id {5f70a987-c0e6-4a5e-98e2-609a7899b6fb}
   Method TrackRaDec: Id {30315973-ed3d-4ebf-826f-7c2c721d63f9} *)
